TEXTLIST TL_SingleAxisJogMode
  0 = 'Standard slow'
  1 = 'Standard fast'
  2 = 'Continous'
  3 = 'Inching'
  4 = 'Inching modulo'
   = ''
END_TEXTLIST

(* stored: Version 1.1.0.1, ProductVersion 3.1.4024.9
   TextList TL_SingleAxisJogMode: Id {43de5411-e4ae-4e98-86f1-8b369d0cfe1b} *)
